# B&R Automation Studio project BR_ZBM1 (part 4)

#### Serial.st
```iecst
(********************************************************************
 * COPYRIGHT -- Microsoft
 ********************************************************************
 * Package: Serial
 * File: Serial.st
 * Author: jorkes
 * Created: November 26, 2014
 *******************************************************************)
FUNCTION_BLOCK fbSerial
	Sender.Commands.open_send := enable;

	CASE Sender.step OF
		FRM_WAIT:	(*--- wait for command*)

			IF Sender.Commands.open_send = TRUE THEN								(*command for sender activation*)
				Sender.step := FRM_OPEN;
			END_IF

		(*close will be requested in step FRM_WRITE*)

		FRM_OPEN:	(*--- open serial interface*)

			(*_parameters for FRM_xopen()*)
			Sender.FRM_xopen_0.enable := TRUE;
			Sender.FRM_xopen_0.device := ADR('IF1');										(*Devicename --> see your serial interface properties*)
			Sender.FRM_xopen_0.mode := ADR('/PHY=RS232 /BD=9600 /DB=8 /PA=N /SB=1'); 		(*Modestring --> specifies the seria operation mode*)
			Sender.FRM_xopen_0.config := ADR(Sender.xopenConfig) ;					(*Additional _parameters, optional*)

			(*Additional _parameters for FRM_xopen()*)
			Sender.xopenConfig.idle := 10;											(*Idle time between two characters*)
			Sender.xopenConfig.delimc := 0;											(*activate two delimeters*)
			Sender.xopenConfig.delim[0] := 0; 										(*CR - carridge return -> dec 13*)
			Sender.xopenConfig.delim[1] := 0; 										(*LF - line feed -> dec 10*)
			Sender.xopenConfig.tx_cnt := 3;											(*number of transmit buffers*)
			Sender.xopenConfig.rx_cnt := 3; 										(*number of receive buffers*)
			Sender.xopenConfig.tx_len := 256; 										(*length of transmit buffers*)
			Sender.xopenConfig.rx_len := 256; 										(*lenght of receive buffers*)
			Sender.xopenConfig.argc := 0;											(*activate additional options*)
			Sender.xopenConfig.argv := 0;											(*_parameters for additional options (check help)*)

			Sender.FRM_xopen_0();													(*call the FRM_xopen() function*)

			IF Sender.FRM_xopen_0.status = 0 THEN
				Sender.step := FRM_GBUF;											(*Interface opend successfully --> next step*)
			ELSIF Sender.FRM_xopen_0.status = BUSY THEN
				Sender.step := FRM_OPEN;											(*operation not finished yet --> call again*)
			ELSE
				Sender.step := FRM_ERROR;											(*function returned errorcode --> check help*)
			END_IF

		FRM_GBUF:	(*--- aquire sendbuffer for FRM_WRITE*)
			Sender.FRM_gbuf_0.enable := TRUE;
			Sender.FRM_gbuf_0.ident := Sender.FRM_xopen_0.ident;

			Sender.FRM_gbuf_0();													(*call the FRM_gbuf() function*)

			IF Sender.FRM_gbuf_0.status = 0 THEN
				memset(Sender.FRM_gbuf_0.buffer,0,Sender.FRM_gbuf_0.buflng);		(*clear sendbuffer*)
				Sender.send_data := text;
				strcpy(Sender.FRM_gbuf_0.buffer,ADR(Sender.send_data));					(*copy senddata to sendbuffer*)
				Sender.FRM_write_0.enable := TRUE;
				Sender.FRM_write_0.ident := Sender.FRM_xopen_0.ident;					(*ident from FRM_xopen()*)
				Sender.FRM_write_0.buffer := Sender.FRM_gbuf_0.buffer;					(*sendbuffer*)
				Sender.FRM_write_0.buflng := strlen(ADR(Sender.send_data));				(*net length of senddata*)

				Sender.FRM_write_0();													(*call the FRM_write() function*)

				IF Sender.FRM_write_0.status = 0 THEN
					IF Sender.Commands.close = TRUE THEN								(*requst to close the serial port*)
						Sender.Commands.open_send := FALSE;								(*disable command open_send*)
						Sender.step := FRM_CLOSE;
					ELSE
						Sender.step := FRM_GBUF;										(*writing successful --> get next sendbuffer*)
					END_IF
				ELSIF NOT Sender.FRM_write_0.status = BUSY THEN
					Sender.step := FRM_ROBUF;											(*function returned errorcode --> check help*)
				END_IF
			END_IF

		FRM_ROBUF:	(*--- release sendbuffer in case of no successful write operation*)
			Sender.FRM_robuf_0.enable := TRUE;
			Sender.FRM_robuf_0.buffer := Sender.FRM_gbuf_0.buffer;					(*sendbuffer*)
			Sender.FRM_robuf_0.buflng := Sender.FRM_gbuf_0.buflng;					(*buffer length*)
			Sender.FRM_robuf_0.ident := Sender.FRM_xopen_0.ident;					(*ident open*)

			Sender.FRM_robuf_0();													(*call the FRM_robuf() function*)

			IF Sender.FRM_robuf_0.status = 0 THEN
				Sender.step := FRM_GBUF;											(*released buffer successful --> get next sendbuffer*)
			ELSIF Sender.FRM_robuf_0.status = BUSY THEN
				Sender.step := FRM_ROBUF;											(*operation not finished yet --> call again*)
			ELSE
				Sender.step := FRM_ERROR;											(*function returned errorcode --> check help*)
			END_IF

		FRM_CLOSE:	(*--- close the interface*)
			Sender.FRM_close_0.enable := TRUE;
			Sender.FRM_close_0.ident := Sender.FRM_xopen_0.ident;					(*ident from FRM_xopen()*)

			Sender.FRM_close_0();													(*call the FRM_close() function*)

			IF Sender.FRM_close_0.status = 0 THEN
				Sender.Commands.close := FALSE;										(*disable close command*)
				Sender.step := FRM_WAIT;											(*closed interface successfully --> wait step*)
			ELSIF Sender.FRM_close_0.status = BUSY THEN
				Sender.step := FRM_CLOSE;											(*operation not finished yet --> call again*)
			ELSE
				Sender.step := FRM_ERROR;											(*function returned errorcode --> check help*)
			END_IF

		FRM_ERROR:	(*--- error handling*)
		; (*not implementet yet, check help for error codes*)
	END_CASE
END_FUNCTION_BLOCK
```

### Library Logical/libraries_hav/SensContr (IEC) - Sensor control library

#### SensContr.fun - Exported functions and function blocks
```iecst
(********************************************************************
 * COPYRIGHT -- Microsoft
 ********************************************************************
 * Library: SensContr
 * File: SensContr.fun
 * Author: jorkes
 * Created: December 01, 2014
 ********************************************************************
 * Functions and function blocks of library SensContr
 ********************************************************************)

FUNCTION_BLOCK fbSensControl
	VAR_INPUT
		IN : BOOL;
		tiSensDelay : TIME;
		tiSensPuls : TIME;
	END_VAR
	VAR_OUTPUT
		Q : BOOL;
	END_VAR
	VAR
		tiTreinDelay : TIME := T#50ms; (*2 x 50ms*)
		tpSensPuls_0 : TP;
		tpSensPuls_1 : TP;
		tpTreinPuls_0 : TP;
		tpTreinPuls_1 : TP;
		zzEdge00000 : BOOL;
		zzEdge00001 : BOOL;
		zzEdge00002 : BOOL;
		zzEdge00003 : BOOL;
	END_VAR
END_FUNCTION_BLOCK

FUNCTION_BLOCK fbSensDelay
	VAR_INPUT
		IN : BOOL;
		tiSensDelay : TIME;
		tiSensPuls : TIME;
	END_VAR
	VAR_OUTPUT
		Q : BOOL;
	END_VAR
	VAR
		tpSensPuls_0 : TP;
		tpSensPuls_1 : TP;
		zzEdge00000 : BOOL;
		zzEdge00001 : BOOL;
	END_VAR
END_FUNCTION_BLOCK
```

#### SensContr.st
```iecst
(********************************************************************
 * COPYRIGHT -- Microsoft
 ********************************************************************
 * Package: SensContr
 * File: SensContr.st
 * Author: jorkes
 * Created: December 01, 2014
 *******************************************************************)
FUNCTION_BLOCK fbSensControl
	tpSensPuls_0(IN := EDGEPOS(IN), PT := tiSensDelay);
	tpSensPuls_1(IN := EDGENEG(tpSensPuls_0.Q), PT := tiSensPuls);
	Q := tpSensPuls_1.Q;
END_FUNCTION_BLOCK
FUNCTION_BLOCK fbSensDelay
	tpSensPuls_0(IN := EDGEPOS(IN), PT := tiSensDelay);
	tpSensPuls_1(IN := EDGENEG(tpSensPuls_0.Q), PT := tiSensPuls);
	Q := tpSensPuls_1.Q;
END_FUNCTION_BLOCK
```

### Library Logical/libraries_hav/MBU_lib (IEC) - Main Belt Unit library

#### MBU_lib.typ - Exported data types
```iecst
(********************************************************************
 * COPYRIGHT -- Microsoft
 ********************************************************************
 * Library: MBU_lib
 * File: MBU_lib.typ
 * Author: jorkes
 * Created: December 01, 2014
 ********************************************************************
 * Data types of library MBU_lib
 ********************************************************************)

TYPE
	enumMBU_CMD :
		(
		MBU_CMD_INIT,
		MBU_CMD_RUN,
		MBU_CMD_STOP,
		MBU_CMD_MANUAL,
		MBU_CMD_FAULT
		);
	enumMBU_ST :
		(
		MBU_ST_INIT,
		MBU_ST_RUN,
		MBU_ST_HOLD,
		MBU_ST_READY,
		MBU_ST_DISABLED,
		MBU_ST_MANUAL,
		MBU_ST_ERROR,
		MBU_ST_SIMULATED
		);
	MBU_Interface : 	STRUCT
		bEnable : BOOL;
		bReset : BOOL;
		bBeltShiftReg : ARRAY[0..39]OF BOOL;
		uiBeltShiftReg1 : UDINT;
		uiBeltShiftReg2 : UDINT;
		usBunchPositions : USINT := 39;
		usAflegPos : USINT := 37;
		usBindPos2 : USINT := 33;
		usBindPos1 : USINT := 31;
		usKnifePos : USINT := 27;
		tiSensPuls : TIME := T#20ms;
		tiBindPuls : TIME := T#100ms;
		tiBindDelay2 : TIME := T#50ms;
		tiBindDelay1 : TIME := T#50ms;
		tiSensDelay2 : TIME := T#70ms; (*Vakkenband*)
		tiSensDelay1 : TIME := T#420ms; (*Sponsband*)
		usMovePositions : USINT := 0;
		bReadyToReceive : BOOL := FALSE;
		bToggleBelt : BOOL := FALSE;
		bToggleKnife : BOOL := FALSE;
		bToggleBuffer : BOOL := FALSE;
		bSimulate : BOOL := FALSE; (*Set high for simulation*)
		bFault : BOOL := FALSE; (*MBU Fault state*)
		Command : enumMBU_CMD := MBU_CMD_STOP;
		State : enumMBU_ST := MBU_ST_HOLD;
		tiKnifePuls : TIME;
		tiBufferPuls : TIME;
		tiBufferDelay : TIME;
	END_STRUCT;
	MainbeltUnit : 	STRUCT  (*Verzameling parameters bosband*)
		in_bMainBeltSensor1 : BOOL := FALSE;
		in_bMainBeltSensor2 : BOOL := FALSE;
		in_bElastiekOp1 : BOOL := FALSE;
		in_bElastiekOp2 : BOOL := FALSE;
		out_bBinder1 : BOOL := FALSE;
		out_bBinder2 : BOOL := FALSE;
		typInterface : MBU_Interface;
		typBeltMotor1 : AcpInverter_typ;
		motBelt1 : ACPinverter;
		typBeltMotor2 : AcpInverter_typ;
		motBelt2 : ACPinverter;
		typMainMotor : AcpInverter_typ;
		motMain : ACPinverter;
		typPreCutter : AcpInverter_typ;
		motPreCutter : ACPinverter;
		typBufferMotor : AcpInverter_typ;
		motBufferBelt : ACPinverter;
		typKnifeUnit : AcpInverter_typ;
		motKnifeUnit : ACPinverter;
	END_STRUCT;
END_TYPE
```

#### MBU_lib.fun - Exported functions and function blocks
```iecst
(********************************************************************
 * COPYRIGHT -- Microsoft
 ********************************************************************
 * Library: MBU_lib
 * File: MBU_lib.fun
 * Author: jorkes
 * Created: December 01, 2014
 ********************************************************************
 * Functions and function blocks of library MBU_lib
 ********************************************************************)

FUNCTION fbShiftBelt : BOOL
	VAR_INPUT
		ThisMBU : MainbeltUnit;
		enable : BOOL;
	END_VAR
	VAR
		idx : USINT;
		size : USINT;
		overflow : UDINT;
	END_VAR
END_FUNCTION

FUNCTION fbCheckBUReadyForDrop : BOOL
	VAR_INPUT
		BU : ARRAY[0..9] OF BunchUnit;
		size : USINT;
	END_VAR
	VAR
		idx : USINT;
		sum : USINT;
	END_VAR
END_FUNCTION

FUNCTION fbCheckBelt : BOOL
	VAR_INPUT
		ThisMBU : MainbeltUnit;
	END_VAR
	VAR
		idx : USINT;
		sum : USINT;
		size : USINT;
	END_VAR
END_FUNCTION

FUNCTION fbHasFlowersOnIndex : BOOL
	VAR_INPUT
		ThisMBU : MainbeltUnit;
		idx : USINT;
	END_VAR
	VAR
		uiMask : UDINT;
		uiOut : UDINT;
	END_VAR
END_FUNCTION

FUNCTION fbSetFlowersOnIndex : BOOL
	VAR_INPUT
		ThisMBU : MainbeltUnit;
		idx : USINT;
		bHasFlower : BOOL;
	END_VAR
	VAR
		uiMask : USINT;
		uiOut : USINT;
	END_VAR
END_FUNCTION
```

#### MBU_lib.st
```iecst
(********************************************************************
 * COPYRIGHT -- Microsoft
 ********************************************************************
 * Package: MBU_lib
 * File: MBU_lib.st
 * Author: jorkes
 * Created: December 01, 2014
 *******************************************************************)

FUNCTION fbShiftBelt
//	size := ( SIZEOF(ThisMBU.typInterface.bBeltShiftReg)/SIZEOF(ThisMBU.typInterface.bBeltShiftReg[0]) );
//
//	IF enable THEN
//		FOR idx := (size - 1) TO 1 BY -1 DO
//			ThisMBU.typInterface.bBeltShiftReg[idx] := ThisMBU.typInterface.bBeltShiftReg[idx-1];
//		END_FOR
//	END_IF
	overflow := SHL(ThisMBU.typInterface.uiBeltShiftReg2,1);
	overflow := SHL(ThisMBU.typInterface.uiBeltShiftReg1,1);
	ThisMBU.typInterface.uiBeltShiftReg2 := ((ThisMBU.typInterface.uiBeltShiftReg2 + overflow) AND 16#00FF); // 32 + 8 postities
	fbShiftBelt := TRUE;
END_FUNCTION

FUNCTION fbCheckBelt
//	size := ( SIZEOF(ThisMBU.typInterface.bBeltShiftReg)/SIZEOF(ThisMBU.typInterface.bBeltShiftReg[0]) );
//
//	sum := 0;
//	FOR idx := 0 TO (size - 1) DO
//		sum := sum + ThisMBU.typInterface.bBeltShiftReg[idx];
//	END_FOR

//	IF sum <> 0 THEN
	IF ThisMBU.typInterface.uiBeltShiftReg1 <> 0 OR ThisMBU.typInterface.uiBeltShiftReg2 <> 0 THEN
		fbCheckBelt := TRUE;
	ELSE
		fbCheckBelt := FALSE;
	END_IF
END_FUNCTION

FUNCTION fbCheckBUReadyForDrop
	// size := 10; Set by caller
	sum := 0;
	FOR idx := 0 TO (size - 1) DO
		sum := sum + BU[idx].typInterface.bReadyForDrop;
	END_FOR

	//memco

	IF sum <> 0 THEN
		fbCheckBUReadyForDrop := TRUE;
	ELSE
		fbCheckBUReadyForDrop := FALSE;
	END_IF
END_FUNCTION

FUNCTION fbHasFlowersOnIndex

//	IF( ThisMBU.typInterface.bBeltShiftReg[idx] ) THEN
//		fbHasFlowersOnIndex := TRUE;
//	ELSE
//		fbHasFlowersOnIndex := FALSE;
//	END_IF
	IF idx <32 THEN
		uiMask :=1;
		uiOut := SHL(uiMask, idx);

		IF( ThisMBU.typInterface.uiBeltShiftReg1 AND uiMask) <> 0 THEN
			fbHasFlowersOnIndex := TRUE;
		ELSE
			fbHasFlowersOnIndex := FALSE;
		END_IF
	ELSE
		uiMask :=1;
		uiOut := SHL(uiMask, idx - 32);

		IF( ThisMBU.typInterface.uiBeltShiftReg2 AND uiMask) <> 0 THEN
			fbHasFlowersOnIndex := TRUE;
		ELSE
			fbHasFlowersOnIndex := FALSE;
		END_IF
	END_IF
END_FUNCTION

FUNCTION fbSetFlowersOnIndex
//	ThisMBU.typInterface.bBeltShiftReg[idx] := bHasFlower;
//	fbSetFlowersOnIndex := TRUE;
	IF idx <32 THEN
		uiMask :=1;
		uiOut := SHL(uiMask, idx);

		ThisMBU.typInterface.uiBeltShiftReg1 := ThisMBU.typInterface.uiBeltShiftReg1 OR uiMask;

	ELSE
		uiMask :=1;
		uiOut := SHL(uiMask, idx - 32);

		ThisMBU.typInterface.uiBeltShiftReg2 := ThisMBU.typInterface.uiBeltShiftReg2 OR uiMask;
	END_IF

END_FUNCTION
```

### Library Logical/libraries_hav/Hardware (IEC) - A new source library

#### Hardware.typ - Exported data types
```iecst
(********************************************************************
 * COPYRIGHT --
 ********************************************************************
 * Library: Hardware
 * File: Hardware.typ
 * Author: ronspa
 * Created: February 03, 2015
 ********************************************************************
 * Data types of library Hardware
 ********************************************************************)

TYPE
	modulTyp : 	STRUCT
		bModuleOK : BOOL;
		uModuleID : UINT;
	END_STRUCT;
END_TYPE
```
